FUNCTION_BLOCK DLOG_DINT_1
VAR_IN_OUT
	X : DLOG_DATA;
END_VAR
VAR_INPUT
	VALUE : DINT;
	COLUMN : STRING(40);
	DELTA : DINT;
END_VAR
VAR
	UCB : UNI_CIRCULAR_BUFFER;
	init : BOOL;
	id : WORD;
	delta_last : DINT;
	value_last : DINT;
END_VAR

(*
version 1.2		25. july. 2011
programmer		ks
tested by			ks

DLOG_DINT legt den DINT-Wert als STRING im FIFO-RING-Buffer ab um diesen mit den Baustein DLOG_STORE_* aufzuzeichnen
*)

IF NOT init THEN
	init := TRUE;
	X.ID_MAX := X.ID_MAX + 1;
	id := WORD#16#0801; (* Quelltype DINT , Zieltype STRING *)
END_IF;

IF X.ADD_HEADER THEN
	X.UCB.D_STRING := COLUMN;
	X.UCB.D_HEAD := id;
	X.UCB.D_MODE := 1;
	UCB(DATA:=X.UCB); (* Daten eintragen *)
ELSIF X.ADD_DATA THEN
	X.UCB.D_STRING := DINT_TO_STRING(value_last);
	X.UCB.D_HEAD := id;
	X.UCB.D_MODE := 1;
	UCB(DATA:=X.UCB); (* Daten eintragen *)
	delta_last := value_last;
ELSIF DELTA <> 0 THEN
	IF VALUE <= (delta_last - DELTA) OR VALUE >= (delta_last + DELTA) THEN
		X.ADD_DATA_REQ := TRUE;
		delta_last := VALUE;
	END_IF;
END_IF;
value_last := VALUE;

(* revision history
ks	01. jan. 2011	rev 1.0
	original version

ks	17. may. 2011	rev 1.1
	DELTA Funktion integriert

ks	25. july.   2011	rev 1.2
	neue head information
*)

END_FUNCTION_BLOCK

(* stored: Version 1.1.0.1, ProductVersion 3.1.4024.0
   POU DLOG_DINT_1: Id {d7d55a23-313e-42dd-80fe-2469ce57de63}, SpecialFunc None *)
